FUNCTION_BLOCK FB_FastClose
VAR_INPUT
    MotorClosedPositionPlus : INT;       // P1 (positive closed)
    C2 : INT;                            // Encoder actual count
    SlitStatusFlagIn : INT;              // Input Df for position check
END_VAR
VAR_IN_OUT
    EncoderShadow : INT;                 // Cs (shadow register)
    SlitStatusFlag : INT;                // Df
END_VAR
VAR_OUTPUT
    Complete : BOOL := FALSE;
END_VAR
VAR
    State : INT := 0; // 0: idle, 1: moving, 2: done
END_VAR

METHOD Execute : BOOL
VAR_INPUT
END_VAR
IF State = 0 THEN
    // Only move if not already closed
    IF (SlitStatusFlagIn <> 1) AND (SlitStatusFlagIn <> -1) THEN
        State := 1;       // Start moving to P1
        Complete := FALSE;
    ELSE
        // Already closed, skip to complete
        State := 2;
        Complete := TRUE;
    END_IF
ELSIF State = 1 THEN
    // Simulate motion complete; check actual axis in a real system
    EncoderShadow := C2;
    SlitStatusFlag := 1;   // Positive closed
    State := 2;
    Complete := TRUE;
END_IF
END_METHOD

METHOD Reset : BOOL
VAR_INPUT
END_VAR
    State := 0;
    Complete := FALSE;
END_METHOD

END_FUNCTION_BLOCK

(* stored: Version 1.1.0.1
   POU FB_FastClose: Id {0e94abec-494d-4612-9922-721fd3573be3}, SpecialFunc None
   Method Execute: Id {8f6e7839-24ed-4da1-9332-4bca9bff8b25}
   Method Reset: Id {7be53d8d-7041-4f2c-9656-99bba48ded5b} *)
